// TIA Portal V19 export
FUNCTION "FC_Optimierung_Pos" : Void   // FC171, STL
{ S7_Optimized_Access := 'TRUE' }
// stored: AutoNumber false
   VAR_INPUT
      Pos : Int;
      Umsetzzeit : DInt;
   END_VAR
   VAR_OUTPUT
      Belegt : Bool;
   END_VAR
   VAR_IN_OUT
      Restzeit : DInt;
   END_VAR
   VAR_TEMP
      WT_DB : Int;
      Cmd : Int;
   END_VAR
BEGIN

NETWORK
TITLE = 
      L     0;
      T     #Restzeit;

      SET;
      R     #Belegt;

      L     0;
      L     "DB_POS".POS[#Pos].next_WT;
      ==I;
      BEC;
      S     #Belegt;
      +     100;
      T     #WT_DB;

      L     0;
      L     "DB_POS".POS[#Pos].WT_DB;
      ==I;
      L     "DB_POS".POS[#Pos].Soll_Expozeit;
      JC    setZ;
      L     "DB_POS".POS[#Pos].Restzeit;
setZ: T     #Restzeit;

      OPN   DB [#WT_DB];
      L     %DBW48;  //"DB_WT1".B_PNTER
retC: T     #Cmd;

      L     %DBW0;  //"DB_WT1".ANZAHL
      >=I;
      JC    ende;

      L     #Cmd;
      L     %DBW4;  //"DB_WT1".LENG
      *D;
      L     %DBW2;  //"DB_WT1".OFFSET
      +D;
      SLD   3;
      LAR1;

      L     #Restzeit;
      L     #Umsetzzeit;
      +D;
      T     #Restzeit;

      L     DBB [AR1, P#1.0];  //"DB_WT1".Befehl[#Cmd].Startpos
      L     18;
      >I;
      JC    ende;

      L     0;
      L     DBW [AR1, P#6.0];  //"DB_WT1".Befehl[#Cmd].Param_Ptr
      ==I;
      JC    nexC;
      SLD   3;
      LAR1;
      L     #Restzeit;
      L     DBD [AR1, P#0.0];
      +D;
      T     #Restzeit;

nexC: L     #Cmd;
      +     1;
      JU    retC;


ende: NOP   0;

END_FUNCTION
